// TIA Portal V19 export
FUNCTION "FC_AMS_304i" : Void   // FC204, STL
TITLE = Absolut-Wegmessung
{ S7_Optimized_Access := 'FALSE' }
// stored: AutoNumber false
   VAR_INPUT
      Eingangswert : DInt;   // kompletter Eingangswert
      LE_Status : Word;   // Status enthält Diodenstatus und Fehler vom Gerät
      FW_Nr : Int;   // Fahrwagen-Nr.
   END_VAR
   VAR_IN_OUT
      Steuerwort : Word;   // Laserdiode ein-/ausschalten
   END_VAR
   VAR_TEMP
      Messung : DInt;   // neuer gemessener Wert
      Messwert : DInt;   // Messwert in mm
      Offset : DInt;
      DB_Nr : Word;
      FW_DB : Word;
      count : Byte;
      Req_Laser : Bool;   // Anforderung Messwert
      invers : Bool;
      Laser_on : Bool;
      Alarm : Bool;
      Warng_Signal : Bool;
      Warng_Temp : Bool;
      Warng_Plausi : Bool;
      Anz_FM : Int;   // Anzahl Fehlmessungen
      Laser_was_on : Bool;
   END_VAR
BEGIN

NETWORK
TITLE = Werte aus FW holen
//----------------------------
// Aufbereitung Eingangswerte
//----------------------------
      L     #FW_Nr;
      L     10;
      +I;
      T     #FW_DB;
      OPN   DB [#FW_DB];
      L     0;
      L     %DBB210;  //"DI_FW_1".PAR.Fahrt.Dir_negativ
      <>I;
      =     #invers;

      L     %DBD206;  //"DI_FW_1".PAR.Fahrt.MessOffset
      T     #Offset;

      A     %DBX70.3;  //"DI_FW_1".OUT.Req_Laser
      =     #Req_Laser;

      A     %DBX51.7;  //"DI_FW_1".IN.Laser_on
      =     #Laser_on;

      L     %DBB211;  //"DI_FW_1".PAR.Fahrt.ErrCount
      T     #Anz_FM;

      L     %DBB361;  //"DI_FW_1".TMP.ErrCount_Possys
      T     #count;

      L     %DBD4;  //"DI_FW_1".ZST.PosInc
      T     #Messwert;


NETWORK
TITLE = 
//----------------------
//Warnungen
//----------------------

      A     #Req_Laser;
      AN    #LE_Status.%X0;  //Laser_off
      AN    #LE_Status.%X4;  //Lasersignal zu gering
      S     #Laser_on;

      AN    #Req_Laser;
      R     #Laser_on;

      A     #LE_Status.%X4;  //Lasersignal zu gering
      A     #Laser_on;
      =     #Warng_Signal;  //Signalpegel zu gering

      A     #LE_Status.%X5;  //Temperatur zu hoch
      =     #Warng_Temp;  //Temperatur zu hoch

      A     #LE_Status.%X7;  //Plausibilität
      A     #Laser_on;
      =     #Warng_Plausi;

      A     #LE_Status.%X4;  //Lasersignal zu gering//
      A     #Laser_on;
      =     #Alarm;

      A     #LE_Status.%X8;  //Harwarefehler
      S     #Alarm;

//----------------------
//Laserdiode steuern
//----------------------
      A     #Req_Laser;
      L     0;
      JC    Las;
      L     16#0100;
Las:  T     #Steuerwort;

//----------------------
//Gerät defekt
//----------------------
      A     #Alarm;
      JC    out;

//----------------------
//Laserdiode aus
//----------------------
      A     #Req_Laser;  //neu falls Diode nicht einschaltet
      O     #Laser_on;
      JC    mess;
      L     0;
      T     #count;
      JU    out;
//-----------------
//    Messwert
//-----------------
mess: L     #Eingangswert;
      T     #Messung;
      L     0;
      >D;
      JC    ok;

      L     #Anz_FM;
      A     #Laser_on;
      JC    chk;
      L     2;
      *I;
chk:  L     #count;
      <=I;
      JC    err;
      +     1;
      T     #count;
      JU    out;
err:  SET;
      S     #Alarm;
      JU    out;

ok:   SET;
      R     #Alarm;

      L     0;
      T     #count;

      L     #Offset;
      L     #Messung;
      A     #invers;
      JC    sub;
      +D;
      T     #Messwert;
      JU    out;

sub:  -D;
      T     #Messwert;
      JU    out;


NETWORK
TITLE = 
out:  OPN   DB [#FW_DB];
      L     #count;
      T     %DBB361;  //"DI_FW_1".TMP.ErrCount_Possys

      L     #Messwert;
      T     %DBD4;  //"DI_FW_1".ZST.PosInc

      A     #Warng_Signal;
      =     %DBX66.0;  //"DI_FW_1".ErrIn.Warnung.Wrn_Optik_PosSys
      A     #Warng_Temp;
      =     %DBX66.1;  //"DI_FW_1".ErrIn.Warnung.Wrn_Temp_PosSys
      A     #Warng_Plausi;
      =     %DBX66.2;  //"DI_FW_1".ErrIn.Warnung.Wrn_Plaus_PosSys
      A     #Alarm;
      =     %DBX62.1;  //"DI_FW_1".ErrIn.Alarm.PosSys
      A     #Laser_on;
      =     %DBX51.7;  //"DI_FW_1".IN.Laser_on

END_FUNCTION
